FUNCTION_BLOCK InfoDataAdsAoE EXTENDS InfoDataAds
VAR
	_AoeNetId AT %I*: AMSNETID;
END_VAR

PROPERTY AdsAddr : AMSADDR
GET
AdsAddr := _AdsAddr;
END_GET
END_PROPERTY

END_FUNCTION_BLOCK

(* stored: Version 1.1.0.1, ProductVersion 3.1.4024.9
   POU InfoDataAdsAoE: Id {de23081f-d2be-0df9-1f69-80946b2efe4b}, SpecialFunc None
   Property AdsAddr: Id {6e681fcc-0d7c-0b0e-0742-088acae6a4e1}
   Get Get: Id {66f4cca1-7574-02cf-0299-10a7217d1ff2} *)
